FUNCTION_BLOCK fb_switchclkcheck
VAR_OUTPUT
	swXgood: BOOL := TRUE;
END_VAR
VAR
	prev_clk: BOOL;
END_VAR

(*This function block sends an alternating signal at a frequency of 100 Hz, and checks whether 
it has been altered from previous check*)

(*
TCout.SwCLK := NOT TCout.SwCLK;	
IF prev_clk = TCout.SwCLK THEN
	swXgood := FALSE;
ELSE 
	swXgood := TRUE;
END_IF
prev_clk := TCout.SwCLK; //only for testing => when doing physical setup => prev_clk := TCin.CollisionSW; 
*)

IF TCin.CollisionSW = FALSE THEN
	// STOP
END_IF

END_FUNCTION_BLOCK

(* stored: Version 1.1.0.1, ProductVersion 3.1.4024.5
   POU fb_switchclkcheck: Id {14220d4d-3f79-4e58-af89-d39b101e9d41}, SpecialFunc None *)
